// TIA Portal V17 export
// export: Created 2025-03-05T08:02:51.1095713Z, ExportSetting WithDefaults, DisplayName Totally Integrated Automation Portal, DisplayVersion V17 Update 8, DisplayName TIA Portal Openness, DisplayVersion V17 Update 8, DisplayName TIA Portal Version Control Interface, DisplayVersion V17, DisplayName SINAMICS Startdrive Advanced, DisplayVersion V17 SP2, DisplayName SINAMICS Startdrive G110M, G120, G120C, G120D, G120P, G115D, DisplayVersion V17 SP2, DisplayName SINAMICS Startdrive G130, G150, S120, S150, SINAMICS MV, S210, DisplayVersion V17 SP2, DisplayName STEP 7 Professional, DisplayVersion V17 Update 8, DisplayName SINUMERIK ONE STEP 7 Toolbox, DisplayVersion V17 Update 12, DisplayName SINUMERIK 840D sl STEP 7 Toolbox, DisplayVersion V17 Update 12, DisplayName STEP 7 Safety, DisplayVersion V17 Update 6, DisplayName WinCC Advanced, DisplayVersion V17 Update 8
FUNCTION "FC7239_HMI_WINCC_OVERVIEW" : Void   // FC7239, LAD
{ S7_Optimized_Access := 'TRUE' }
VERSION : 0.1
// stored: AutoNumber false, IsIECCheckEnabled false, SetENOAutomatically false, UDAEnableTagReadback false
BEGIN

REGION Network 1: UNIT 01 POWDER FEEDER 1 OK
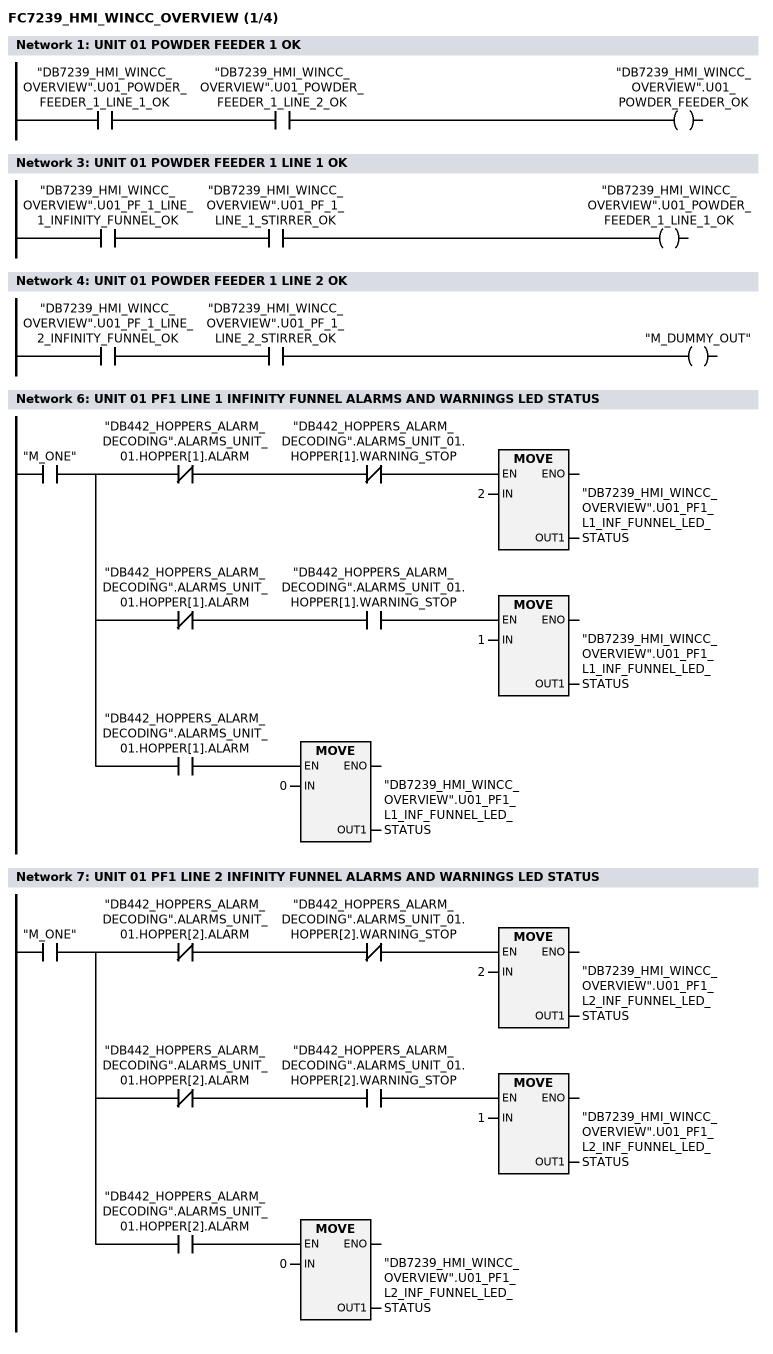
   RUNG wire#powerrail
      Contact( "DB7239_HMI_WINCC_OVERVIEW".U01_POWDER_FEEDER_1_LINE_1_OK )
      Contact( "DB7239_HMI_WINCC_OVERVIEW".U01_POWDER_FEEDER_1_LINE_2_OK )
      Coil( "DB7239_HMI_WINCC_OVERVIEW".U01_POWDER_FEEDER_OK )
   END_RUNG
   // the same network as SCL:
   "DB7239_HMI_WINCC_OVERVIEW".U01_POWDER_FEEDER_OK := "DB7239_HMI_WINCC_OVERVIEW".U01_POWDER_FEEDER_1_LINE_1_OK AND "DB7239_HMI_WINCC_OVERVIEW".U01_POWDER_FEEDER_1_LINE_2_OK;
END_REGION

REGION Network 2: UNIT 02 POWDER FEEDER 2 OK
END_REGION

REGION Network 3: UNIT 01 POWDER FEEDER 1 LINE 1 OK
   RUNG wire#powerrail
      Contact( "DB7239_HMI_WINCC_OVERVIEW".U01_PF_1_LINE_1_INFINITY_FUNNEL_OK )
      Contact( "DB7239_HMI_WINCC_OVERVIEW".U01_PF_1_LINE_1_STIRRER_OK )
      Coil( "DB7239_HMI_WINCC_OVERVIEW".U01_POWDER_FEEDER_1_LINE_1_OK )
   END_RUNG
   // the same network as SCL:
   "DB7239_HMI_WINCC_OVERVIEW".U01_POWDER_FEEDER_1_LINE_1_OK := "DB7239_HMI_WINCC_OVERVIEW".U01_PF_1_LINE_1_INFINITY_FUNNEL_OK AND "DB7239_HMI_WINCC_OVERVIEW".U01_PF_1_LINE_1_STIRRER_OK;
END_REGION

REGION Network 4: UNIT 01 POWDER FEEDER 1 LINE 2 OK
   RUNG wire#powerrail
      Contact( "DB7239_HMI_WINCC_OVERVIEW".U01_PF_1_LINE_2_INFINITY_FUNNEL_OK )
      Contact( "DB7239_HMI_WINCC_OVERVIEW".U01_PF_1_LINE_2_STIRRER_OK )
      Coil( "M_DUMMY_OUT" )
   END_RUNG
   // the same network as SCL:
   "M_DUMMY_OUT" := "DB7239_HMI_WINCC_OVERVIEW".U01_PF_1_LINE_2_INFINITY_FUNNEL_OK AND "DB7239_HMI_WINCC_OVERVIEW".U01_PF_1_LINE_2_STIRRER_OK;
END_REGION

REGION Network 5: <<<<<<<<<<<<<<<<<<<<<<<< UNIT 01 >>>>>>>>>>>>>>>>>>>>>>>>
END_REGION

REGION Network 6: UNIT 01 PF1 LINE 1 INFINITY FUNNEL ALARMS AND WARNINGS LED STATUS
   RUNG wire#powerrail
      Contact( "M_ONE" )
      wire#w1
      I_Contact( "DB442_HOPPERS_ALARM_DECODING".ALARMS_UNIT_01.HOPPER[1].ALARM )
      I_Contact( "DB442_HOPPERS_ALARM_DECODING".ALARMS_UNIT_01.HOPPER[1].WARNING_STOP )
      { S7_GenerateENO := "TRUE" } Move(in := 2, out1 => "DB7239_HMI_WINCC_OVERVIEW".U01_PF1_L1_INF_FUNNEL_LED_STATUS)
   END_RUNG
   RUNG wire#w1
      I_Contact( "DB442_HOPPERS_ALARM_DECODING".ALARMS_UNIT_01.HOPPER[1].ALARM )
      Contact( "DB442_HOPPERS_ALARM_DECODING".ALARMS_UNIT_01.HOPPER[1].WARNING_STOP )
      { S7_GenerateENO := "TRUE" } Move(in := 1, out1 => "DB7239_HMI_WINCC_OVERVIEW".U01_PF1_L1_INF_FUNNEL_LED_STATUS)
   END_RUNG
   RUNG wire#w1
      Contact( "DB442_HOPPERS_ALARM_DECODING".ALARMS_UNIT_01.HOPPER[1].ALARM )
      { S7_GenerateENO := "TRUE" } Move(in := 0, out1 => "DB7239_HMI_WINCC_OVERVIEW".U01_PF1_L1_INF_FUNNEL_LED_STATUS)
   END_RUNG
   // the same network as SCL:
   IF "M_ONE" AND NOT "DB442_HOPPERS_ALARM_DECODING".ALARMS_UNIT_01.HOPPER[1].ALARM AND NOT "DB442_HOPPERS_ALARM_DECODING".ALARMS_UNIT_01.HOPPER[1].WARNING_STOP THEN
       "DB7239_HMI_WINCC_OVERVIEW".U01_PF1_L1_INF_FUNNEL_LED_STATUS := 2;
   END_IF;
   IF "M_ONE" AND NOT "DB442_HOPPERS_ALARM_DECODING".ALARMS_UNIT_01.HOPPER[1].ALARM AND "DB442_HOPPERS_ALARM_DECODING".ALARMS_UNIT_01.HOPPER[1].WARNING_STOP THEN
       "DB7239_HMI_WINCC_OVERVIEW".U01_PF1_L1_INF_FUNNEL_LED_STATUS := 1;
   END_IF;
   IF "M_ONE" AND "DB442_HOPPERS_ALARM_DECODING".ALARMS_UNIT_01.HOPPER[1].ALARM THEN
       "DB7239_HMI_WINCC_OVERVIEW".U01_PF1_L1_INF_FUNNEL_LED_STATUS := 0;
   END_IF;
END_REGION

REGION Network 7: UNIT 01 PF1 LINE 2 INFINITY FUNNEL ALARMS AND WARNINGS LED STATUS
   RUNG wire#powerrail
      Contact( "M_ONE" )
      wire#w1
      I_Contact( "DB442_HOPPERS_ALARM_DECODING".ALARMS_UNIT_01.HOPPER[2].ALARM )
      I_Contact( "DB442_HOPPERS_ALARM_DECODING".ALARMS_UNIT_01.HOPPER[2].WARNING_STOP )
      { S7_GenerateENO := "TRUE" } Move(in := 2, out1 => "DB7239_HMI_WINCC_OVERVIEW".U01_PF1_L2_INF_FUNNEL_LED_STATUS)
   END_RUNG
   RUNG wire#w1
      I_Contact( "DB442_HOPPERS_ALARM_DECODING".ALARMS_UNIT_01.HOPPER[2].ALARM )
      Contact( "DB442_HOPPERS_ALARM_DECODING".ALARMS_UNIT_01.HOPPER[2].WARNING_STOP )
      { S7_GenerateENO := "TRUE" } Move(in := 1, out1 => "DB7239_HMI_WINCC_OVERVIEW".U01_PF1_L2_INF_FUNNEL_LED_STATUS)
   END_RUNG
   RUNG wire#w1
      Contact( "DB442_HOPPERS_ALARM_DECODING".ALARMS_UNIT_01.HOPPER[2].ALARM )
      { S7_GenerateENO := "TRUE" } Move(in := 0, out1 => "DB7239_HMI_WINCC_OVERVIEW".U01_PF1_L2_INF_FUNNEL_LED_STATUS)
   END_RUNG
   // the same network as SCL:
   IF "M_ONE" AND NOT "DB442_HOPPERS_ALARM_DECODING".ALARMS_UNIT_01.HOPPER[2].ALARM AND NOT "DB442_HOPPERS_ALARM_DECODING".ALARMS_UNIT_01.HOPPER[2].WARNING_STOP THEN
       "DB7239_HMI_WINCC_OVERVIEW".U01_PF1_L2_INF_FUNNEL_LED_STATUS := 2;
   END_IF;
   IF "M_ONE" AND NOT "DB442_HOPPERS_ALARM_DECODING".ALARMS_UNIT_01.HOPPER[2].ALARM AND "DB442_HOPPERS_ALARM_DECODING".ALARMS_UNIT_01.HOPPER[2].WARNING_STOP THEN
       "DB7239_HMI_WINCC_OVERVIEW".U01_PF1_L2_INF_FUNNEL_LED_STATUS := 1;
   END_IF;
   IF "M_ONE" AND "DB442_HOPPERS_ALARM_DECODING".ALARMS_UNIT_01.HOPPER[2].ALARM THEN
       "DB7239_HMI_WINCC_OVERVIEW".U01_PF1_L2_INF_FUNNEL_LED_STATUS := 0;
   END_IF;
END_REGION

REGION Network 8: UNIT 01 POWDER LED STATUS
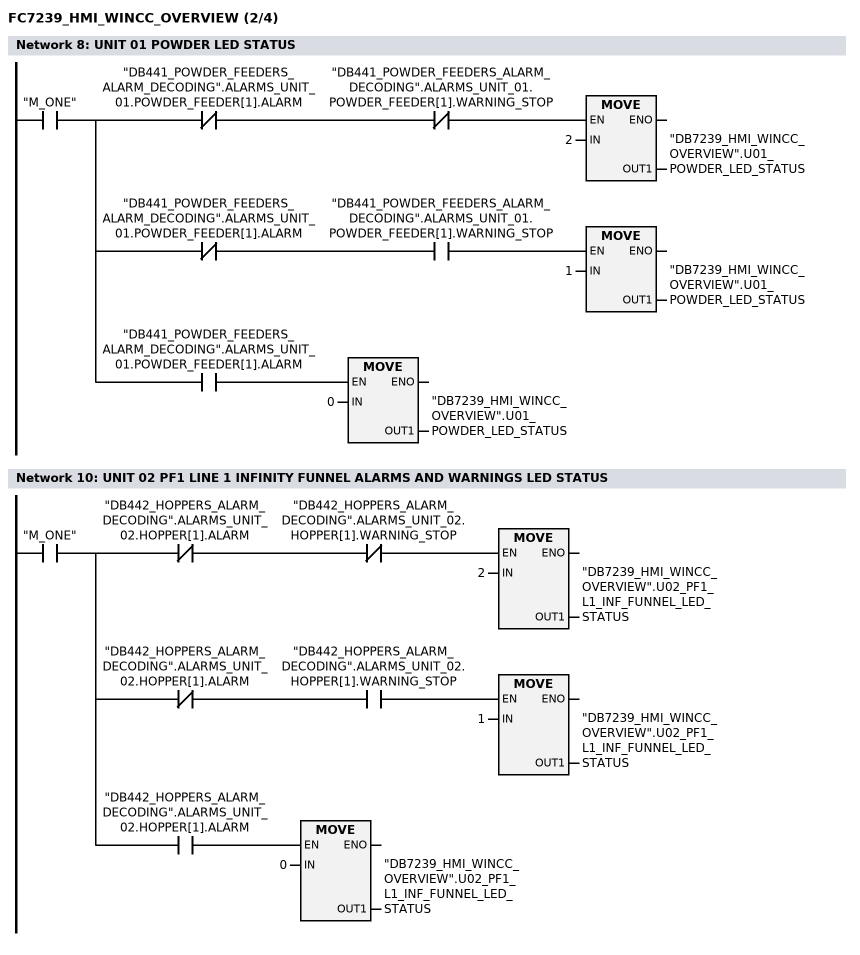
   RUNG wire#powerrail
      Contact( "M_ONE" )
      wire#w1
      I_Contact( "DB441_POWDER_FEEDERS_ALARM_DECODING".ALARMS_UNIT_01.POWDER_FEEDER[1].ALARM )
      I_Contact( "DB441_POWDER_FEEDERS_ALARM_DECODING".ALARMS_UNIT_01.POWDER_FEEDER[1].WARNING_STOP )
      { S7_GenerateENO := "TRUE" } Move(in := 2, out1 => "DB7239_HMI_WINCC_OVERVIEW".U01_POWDER_LED_STATUS)
   END_RUNG
   RUNG wire#w1
      I_Contact( "DB441_POWDER_FEEDERS_ALARM_DECODING".ALARMS_UNIT_01.POWDER_FEEDER[1].ALARM )
      Contact( "DB441_POWDER_FEEDERS_ALARM_DECODING".ALARMS_UNIT_01.POWDER_FEEDER[1].WARNING_STOP )
      { S7_GenerateENO := "TRUE" } Move(in := 1, out1 => "DB7239_HMI_WINCC_OVERVIEW".U01_POWDER_LED_STATUS)
   END_RUNG
   RUNG wire#w1
      Contact( "DB441_POWDER_FEEDERS_ALARM_DECODING".ALARMS_UNIT_01.POWDER_FEEDER[1].ALARM )
      { S7_GenerateENO := "TRUE" } Move(in := 0, out1 => "DB7239_HMI_WINCC_OVERVIEW".U01_POWDER_LED_STATUS)
   END_RUNG
   // the same network as SCL:
   IF "M_ONE" AND NOT "DB441_POWDER_FEEDERS_ALARM_DECODING".ALARMS_UNIT_01.POWDER_FEEDER[1].ALARM AND NOT "DB441_POWDER_FEEDERS_ALARM_DECODING".ALARMS_UNIT_01.POWDER_FEEDER[1].WARNING_STOP THEN
       "DB7239_HMI_WINCC_OVERVIEW".U01_POWDER_LED_STATUS := 2;
   END_IF;
   IF "M_ONE" AND NOT "DB441_POWDER_FEEDERS_ALARM_DECODING".ALARMS_UNIT_01.POWDER_FEEDER[1].ALARM AND "DB441_POWDER_FEEDERS_ALARM_DECODING".ALARMS_UNIT_01.POWDER_FEEDER[1].WARNING_STOP THEN
       "DB7239_HMI_WINCC_OVERVIEW".U01_POWDER_LED_STATUS := 1;
   END_IF;
   IF "M_ONE" AND "DB441_POWDER_FEEDERS_ALARM_DECODING".ALARMS_UNIT_01.POWDER_FEEDER[1].ALARM THEN
       "DB7239_HMI_WINCC_OVERVIEW".U01_POWDER_LED_STATUS := 0;
   END_IF;
END_REGION

REGION Network 9: <<<<<<<<<<<<<<<<<<<<<<<< UNIT 02 >>>>>>>>>>>>>>>>>>>>>>>>
END_REGION

REGION Network 10: UNIT 02 PF1 LINE 1 INFINITY FUNNEL ALARMS AND WARNINGS LED STATUS
   RUNG wire#powerrail
      Contact( "M_ONE" )
      wire#w1
      I_Contact( "DB442_HOPPERS_ALARM_DECODING".ALARMS_UNIT_02.HOPPER[1].ALARM )
      I_Contact( "DB442_HOPPERS_ALARM_DECODING".ALARMS_UNIT_02.HOPPER[1].WARNING_STOP )
      { S7_GenerateENO := "TRUE" } Move(in := 2, out1 => "DB7239_HMI_WINCC_OVERVIEW".U02_PF1_L1_INF_FUNNEL_LED_STATUS)
   END_RUNG
   RUNG wire#w1
      I_Contact( "DB442_HOPPERS_ALARM_DECODING".ALARMS_UNIT_02.HOPPER[1].ALARM )
      Contact( "DB442_HOPPERS_ALARM_DECODING".ALARMS_UNIT_02.HOPPER[1].WARNING_STOP )
      { S7_GenerateENO := "TRUE" } Move(in := 1, out1 => "DB7239_HMI_WINCC_OVERVIEW".U02_PF1_L1_INF_FUNNEL_LED_STATUS)
   END_RUNG
   RUNG wire#w1
      Contact( "DB442_HOPPERS_ALARM_DECODING".ALARMS_UNIT_02.HOPPER[1].ALARM )
      { S7_GenerateENO := "TRUE" } Move(in := 0, out1 => "DB7239_HMI_WINCC_OVERVIEW".U02_PF1_L1_INF_FUNNEL_LED_STATUS)
   END_RUNG
   // the same network as SCL:
   IF "M_ONE" AND NOT "DB442_HOPPERS_ALARM_DECODING".ALARMS_UNIT_02.HOPPER[1].ALARM AND NOT "DB442_HOPPERS_ALARM_DECODING".ALARMS_UNIT_02.HOPPER[1].WARNING_STOP THEN
       "DB7239_HMI_WINCC_OVERVIEW".U02_PF1_L1_INF_FUNNEL_LED_STATUS := 2;
   END_IF;
   IF "M_ONE" AND NOT "DB442_HOPPERS_ALARM_DECODING".ALARMS_UNIT_02.HOPPER[1].ALARM AND "DB442_HOPPERS_ALARM_DECODING".ALARMS_UNIT_02.HOPPER[1].WARNING_STOP THEN
       "DB7239_HMI_WINCC_OVERVIEW".U02_PF1_L1_INF_FUNNEL_LED_STATUS := 1;
   END_IF;
   IF "M_ONE" AND "DB442_HOPPERS_ALARM_DECODING".ALARMS_UNIT_02.HOPPER[1].ALARM THEN
       "DB7239_HMI_WINCC_OVERVIEW".U02_PF1_L1_INF_FUNNEL_LED_STATUS := 0;
   END_IF;
END_REGION

REGION Network 11: UNIT 02 PF1 LINE 2 INFINITY FUNNEL ALARMS AND WARNINGS LED STATUS
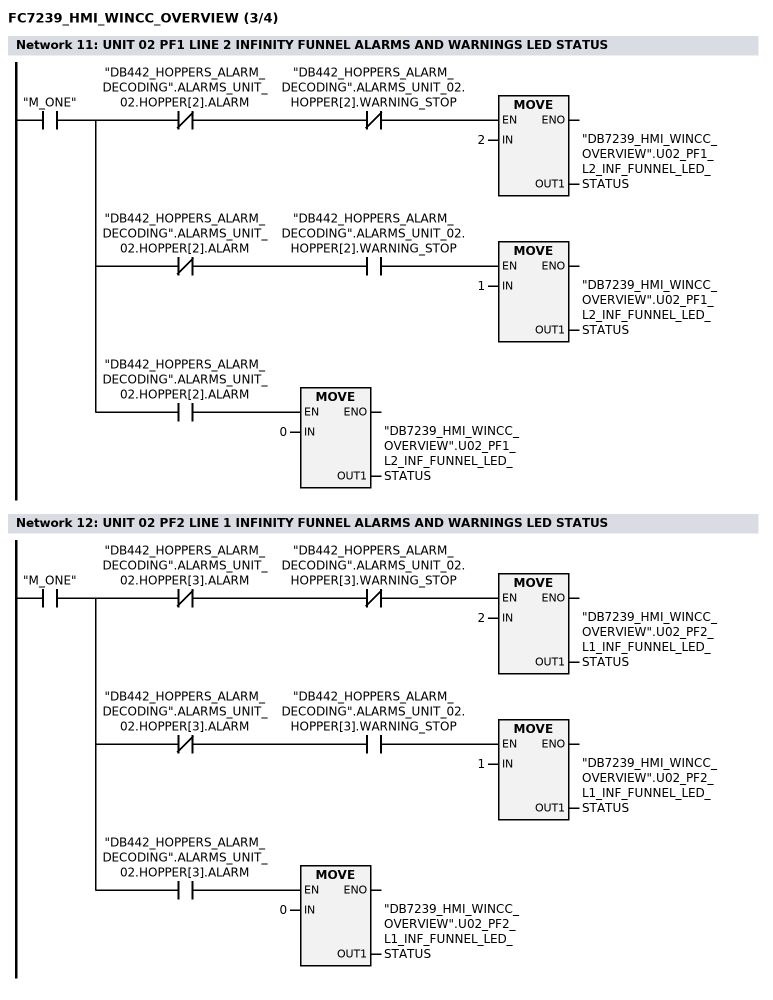
   RUNG wire#powerrail
      Contact( "M_ONE" )
      wire#w1
      I_Contact( "DB442_HOPPERS_ALARM_DECODING".ALARMS_UNIT_02.HOPPER[2].ALARM )
      I_Contact( "DB442_HOPPERS_ALARM_DECODING".ALARMS_UNIT_02.HOPPER[2].WARNING_STOP )
      { S7_GenerateENO := "TRUE" } Move(in := 2, out1 => "DB7239_HMI_WINCC_OVERVIEW".U02_PF1_L2_INF_FUNNEL_LED_STATUS)
   END_RUNG
   RUNG wire#w1
      I_Contact( "DB442_HOPPERS_ALARM_DECODING".ALARMS_UNIT_02.HOPPER[2].ALARM )
      Contact( "DB442_HOPPERS_ALARM_DECODING".ALARMS_UNIT_02.HOPPER[2].WARNING_STOP )
      { S7_GenerateENO := "TRUE" } Move(in := 1, out1 => "DB7239_HMI_WINCC_OVERVIEW".U02_PF1_L2_INF_FUNNEL_LED_STATUS)
   END_RUNG
   RUNG wire#w1
      Contact( "DB442_HOPPERS_ALARM_DECODING".ALARMS_UNIT_02.HOPPER[2].ALARM )
      { S7_GenerateENO := "TRUE" } Move(in := 0, out1 => "DB7239_HMI_WINCC_OVERVIEW".U02_PF1_L2_INF_FUNNEL_LED_STATUS)
   END_RUNG
   // the same network as SCL:
   IF "M_ONE" AND NOT "DB442_HOPPERS_ALARM_DECODING".ALARMS_UNIT_02.HOPPER[2].ALARM AND NOT "DB442_HOPPERS_ALARM_DECODING".ALARMS_UNIT_02.HOPPER[2].WARNING_STOP THEN
       "DB7239_HMI_WINCC_OVERVIEW".U02_PF1_L2_INF_FUNNEL_LED_STATUS := 2;
   END_IF;
   IF "M_ONE" AND NOT "DB442_HOPPERS_ALARM_DECODING".ALARMS_UNIT_02.HOPPER[2].ALARM AND "DB442_HOPPERS_ALARM_DECODING".ALARMS_UNIT_02.HOPPER[2].WARNING_STOP THEN
       "DB7239_HMI_WINCC_OVERVIEW".U02_PF1_L2_INF_FUNNEL_LED_STATUS := 1;
   END_IF;
   IF "M_ONE" AND "DB442_HOPPERS_ALARM_DECODING".ALARMS_UNIT_02.HOPPER[2].ALARM THEN
       "DB7239_HMI_WINCC_OVERVIEW".U02_PF1_L2_INF_FUNNEL_LED_STATUS := 0;
   END_IF;
END_REGION

REGION Network 12: UNIT 02 PF2 LINE 1 INFINITY FUNNEL ALARMS AND WARNINGS LED STATUS
   RUNG wire#powerrail
      Contact( "M_ONE" )
      wire#w1
      I_Contact( "DB442_HOPPERS_ALARM_DECODING".ALARMS_UNIT_02.HOPPER[3].ALARM )
      I_Contact( "DB442_HOPPERS_ALARM_DECODING".ALARMS_UNIT_02.HOPPER[3].WARNING_STOP )
      { S7_GenerateENO := "TRUE" } Move(in := 2, out1 => "DB7239_HMI_WINCC_OVERVIEW".U02_PF2_L1_INF_FUNNEL_LED_STATUS)
   END_RUNG
   RUNG wire#w1
      I_Contact( "DB442_HOPPERS_ALARM_DECODING".ALARMS_UNIT_02.HOPPER[3].ALARM )
      Contact( "DB442_HOPPERS_ALARM_DECODING".ALARMS_UNIT_02.HOPPER[3].WARNING_STOP )
      { S7_GenerateENO := "TRUE" } Move(in := 1, out1 => "DB7239_HMI_WINCC_OVERVIEW".U02_PF2_L1_INF_FUNNEL_LED_STATUS)
   END_RUNG
   RUNG wire#w1
      Contact( "DB442_HOPPERS_ALARM_DECODING".ALARMS_UNIT_02.HOPPER[3].ALARM )
      { S7_GenerateENO := "TRUE" } Move(in := 0, out1 => "DB7239_HMI_WINCC_OVERVIEW".U02_PF2_L1_INF_FUNNEL_LED_STATUS)
   END_RUNG
   // the same network as SCL:
   IF "M_ONE" AND NOT "DB442_HOPPERS_ALARM_DECODING".ALARMS_UNIT_02.HOPPER[3].ALARM AND NOT "DB442_HOPPERS_ALARM_DECODING".ALARMS_UNIT_02.HOPPER[3].WARNING_STOP THEN
       "DB7239_HMI_WINCC_OVERVIEW".U02_PF2_L1_INF_FUNNEL_LED_STATUS := 2;
   END_IF;
   IF "M_ONE" AND NOT "DB442_HOPPERS_ALARM_DECODING".ALARMS_UNIT_02.HOPPER[3].ALARM AND "DB442_HOPPERS_ALARM_DECODING".ALARMS_UNIT_02.HOPPER[3].WARNING_STOP THEN
       "DB7239_HMI_WINCC_OVERVIEW".U02_PF2_L1_INF_FUNNEL_LED_STATUS := 1;
   END_IF;
   IF "M_ONE" AND "DB442_HOPPERS_ALARM_DECODING".ALARMS_UNIT_02.HOPPER[3].ALARM THEN
       "DB7239_HMI_WINCC_OVERVIEW".U02_PF2_L1_INF_FUNNEL_LED_STATUS := 0;
   END_IF;
END_REGION

REGION Network 13: UNIT 02 POWDER LED STATUS
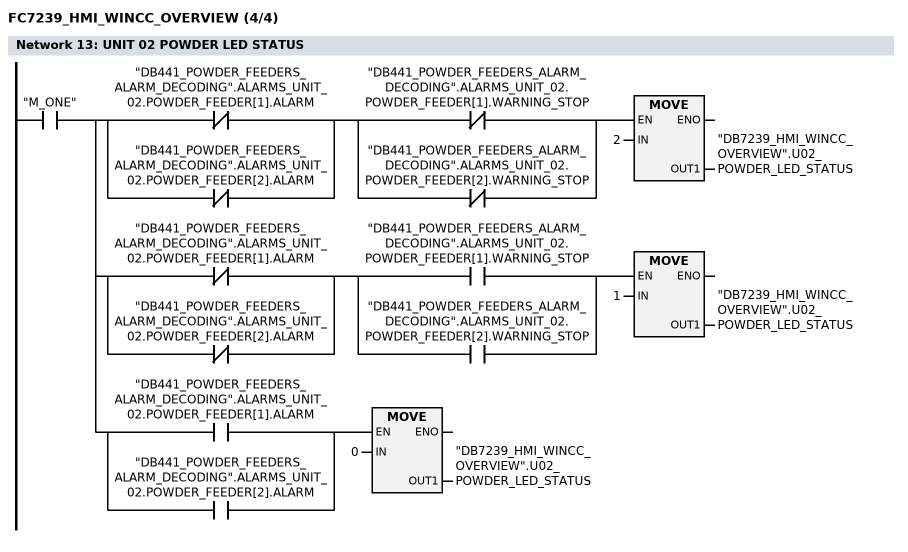
   RUNG wire#powerrail
      Contact( "M_ONE" )
      wire#w1
      I_Contact( "DB441_POWDER_FEEDERS_ALARM_DECODING".ALARMS_UNIT_02.POWDER_FEEDER[1].ALARM )
      wire#w2
      I_Contact( "DB441_POWDER_FEEDERS_ALARM_DECODING".ALARMS_UNIT_02.POWDER_FEEDER[1].WARNING_STOP )
      wire#w3
      { S7_GenerateENO := "TRUE" } Move(in := 2, out1 => "DB7239_HMI_WINCC_OVERVIEW".U02_POWDER_LED_STATUS)
   END_RUNG
   RUNG wire#w1
      I_Contact( "DB441_POWDER_FEEDERS_ALARM_DECODING".ALARMS_UNIT_02.POWDER_FEEDER[2].ALARM )
   END_RUNG wire#w2
   RUNG wire#w2
      I_Contact( "DB441_POWDER_FEEDERS_ALARM_DECODING".ALARMS_UNIT_02.POWDER_FEEDER[2].WARNING_STOP )
   END_RUNG wire#w3
   RUNG wire#w1
      I_Contact( "DB441_POWDER_FEEDERS_ALARM_DECODING".ALARMS_UNIT_02.POWDER_FEEDER[1].ALARM )
      wire#w4
      Contact( "DB441_POWDER_FEEDERS_ALARM_DECODING".ALARMS_UNIT_02.POWDER_FEEDER[1].WARNING_STOP )
      wire#w5
      { S7_GenerateENO := "TRUE" } Move(in := 1, out1 => "DB7239_HMI_WINCC_OVERVIEW".U02_POWDER_LED_STATUS)
   END_RUNG
   RUNG wire#w1
      I_Contact( "DB441_POWDER_FEEDERS_ALARM_DECODING".ALARMS_UNIT_02.POWDER_FEEDER[2].ALARM )
   END_RUNG wire#w4
   RUNG wire#w4
      Contact( "DB441_POWDER_FEEDERS_ALARM_DECODING".ALARMS_UNIT_02.POWDER_FEEDER[2].WARNING_STOP )
   END_RUNG wire#w5
   RUNG wire#w1
      Contact( "DB441_POWDER_FEEDERS_ALARM_DECODING".ALARMS_UNIT_02.POWDER_FEEDER[1].ALARM )
      wire#w6
      { S7_GenerateENO := "TRUE" } Move(in := 0, out1 => "DB7239_HMI_WINCC_OVERVIEW".U02_POWDER_LED_STATUS)
   END_RUNG
   RUNG wire#w1
      Contact( "DB441_POWDER_FEEDERS_ALARM_DECODING".ALARMS_UNIT_02.POWDER_FEEDER[2].ALARM )
   END_RUNG wire#w6
   // the same network as SCL:
   IF "M_ONE" AND (NOT "DB441_POWDER_FEEDERS_ALARM_DECODING".ALARMS_UNIT_02.POWDER_FEEDER[1].ALARM OR NOT "DB441_POWDER_FEEDERS_ALARM_DECODING".ALARMS_UNIT_02.POWDER_FEEDER[2].ALARM) AND (NOT "DB441_POWDER_FEEDERS_ALARM_DECODING".ALARMS_UNIT_02.POWDER_FEEDER[1].WARNING_STOP OR NOT "DB441_POWDER_FEEDERS_ALARM_DECODING".ALARMS_UNIT_02.POWDER_FEEDER[2].WARNING_STOP) THEN
       "DB7239_HMI_WINCC_OVERVIEW".U02_POWDER_LED_STATUS := 2;
   END_IF;
   IF "M_ONE" AND (NOT "DB441_POWDER_FEEDERS_ALARM_DECODING".ALARMS_UNIT_02.POWDER_FEEDER[1].ALARM OR NOT "DB441_POWDER_FEEDERS_ALARM_DECODING".ALARMS_UNIT_02.POWDER_FEEDER[2].ALARM) AND ("DB441_POWDER_FEEDERS_ALARM_DECODING".ALARMS_UNIT_02.POWDER_FEEDER[1].WARNING_STOP OR "DB441_POWDER_FEEDERS_ALARM_DECODING".ALARMS_UNIT_02.POWDER_FEEDER[2].WARNING_STOP) THEN
       "DB7239_HMI_WINCC_OVERVIEW".U02_POWDER_LED_STATUS := 1;
   END_IF;
   IF "M_ONE" AND ("DB441_POWDER_FEEDERS_ALARM_DECODING".ALARMS_UNIT_02.POWDER_FEEDER[1].ALARM OR "DB441_POWDER_FEEDERS_ALARM_DECODING".ALARMS_UNIT_02.POWDER_FEEDER[2].ALARM) THEN
       "DB7239_HMI_WINCC_OVERVIEW".U02_POWDER_LED_STATUS := 0;
   END_IF;
END_REGION
END_FUNCTION
